PROGRAM OK_Repartiteurs_Laser
VAR
	B_820REP1: FB_Rep_Ethercat_MURR;
	B_821REP1: FB_Rep_Ethercat_MURR;
	B_822REP1: FB_Rep_Ethercat_MURR;
	Bandeaux_Leds: FB_LED_LC25C;
	Mesure_Presseur_Aval_Ref: FB_IOLink_Leuze_ODT3CL1;
	Mesure_Presseur_Aval_Opp_Ref: FB_IOLink_Leuze_ODT3CL1;
	Mesure_Presseur_Amont_Ref: FB_IOLink_Leuze_ODT3CL1;
	Mesure_Presseur_Amont_Opp_Ref: FB_IOLink_Leuze_ODT3CL1;
	FB_Servovanne_Gaz_TeteLaser: FB_IOLink_Servo_ITV2030;
	
	Txt_Alarme_Vanne,
	Txt_Defaut_Vanne	:STRING;
	
	Verrine_Machine			:FB_LED_LC25C;

	ReserveIOLink	:BOOL;
	
END_VAR

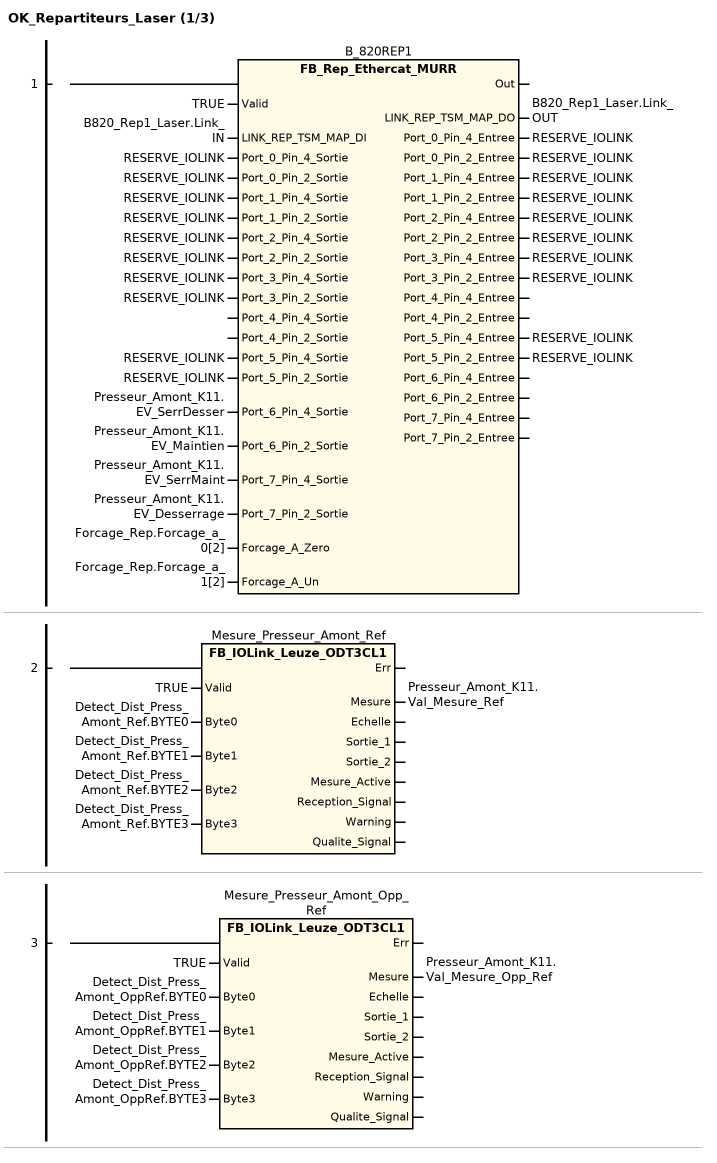
// NETWORK 1
B_820REP1(
    Valid := TRUE,
    LINK_REP_TSM_MAP_DI := B820_Rep1_Laser.Link_IN,
    Port_0_Pin_4_Sortie := RESERVE_IOLINK,
    Port_0_Pin_2_Sortie := RESERVE_IOLINK,
    Port_1_Pin_4_Sortie := RESERVE_IOLINK,
    Port_1_Pin_2_Sortie := RESERVE_IOLINK,
    Port_2_Pin_4_Sortie := RESERVE_IOLINK,
    Port_2_Pin_2_Sortie := RESERVE_IOLINK,
    Port_3_Pin_4_Sortie := RESERVE_IOLINK,
    Port_3_Pin_2_Sortie := RESERVE_IOLINK,
    Port_5_Pin_4_Sortie := RESERVE_IOLINK,
    Port_5_Pin_2_Sortie := RESERVE_IOLINK,
    Port_6_Pin_4_Sortie := Presseur_Amont_K11.EV_SerrDesser,
    Port_6_Pin_2_Sortie := Presseur_Amont_K11.EV_Maintien,
    Port_7_Pin_4_Sortie := Presseur_Amont_K11.EV_SerrMaint,
    Port_7_Pin_2_Sortie := Presseur_Amont_K11.EV_Desserrage,
    Forcage_A_Zero := Forcage_Rep.Forcage_a_0[2],
    Forcage_A_Un := Forcage_Rep.Forcage_a_1[2],
    LINK_REP_TSM_MAP_DO => B820_Rep1_Laser.Link_OUT,
    Port_0_Pin_4_Entree => RESERVE_IOLINK,
    Port_0_Pin_2_Entree => RESERVE_IOLINK,
    Port_1_Pin_4_Entree => RESERVE_IOLINK,
    Port_1_Pin_2_Entree => RESERVE_IOLINK,
    Port_2_Pin_4_Entree => RESERVE_IOLINK,
    Port_2_Pin_2_Entree => RESERVE_IOLINK,
    Port_3_Pin_4_Entree => RESERVE_IOLINK,
    Port_3_Pin_2_Entree => RESERVE_IOLINK,
    Port_5_Pin_4_Entree => RESERVE_IOLINK,
    Port_5_Pin_2_Entree => RESERVE_IOLINK); // FB_Rep_Ethercat_MURR

// NETWORK 2
Mesure_Presseur_Amont_Ref(
    Valid := TRUE,
    Byte0 := Detect_Dist_Press_Amont_Ref.BYTE0,
    Byte1 := Detect_Dist_Press_Amont_Ref.BYTE1,
    Byte2 := Detect_Dist_Press_Amont_Ref.BYTE2,
    Byte3 := Detect_Dist_Press_Amont_Ref.BYTE3,
    Mesure => Presseur_Amont_K11.Val_Mesure_Ref); // FB_IOLink_Leuze_ODT3CL1

// NETWORK 3
Mesure_Presseur_Amont_Opp_Ref(
    Valid := TRUE,
    Byte0 := Detect_Dist_Press_Amont_OppRef.BYTE0,
    Byte1 := Detect_Dist_Press_Amont_OppRef.BYTE1,
    Byte2 := Detect_Dist_Press_Amont_OppRef.BYTE2,
    Byte3 := Detect_Dist_Press_Amont_OppRef.BYTE3,
    Mesure => Presseur_Amont_K11.Val_Mesure_Opp_Ref); // FB_IOLink_Leuze_ODT3CL1

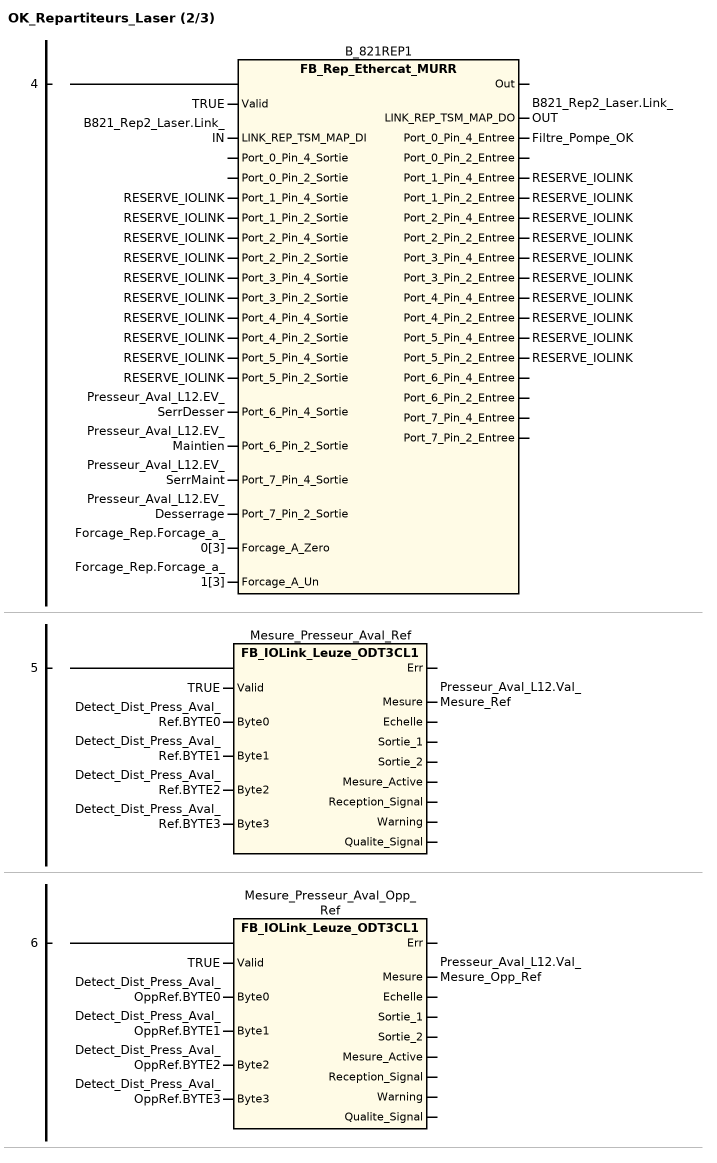
// NETWORK 4
B_821REP1(
    Valid := TRUE,
    LINK_REP_TSM_MAP_DI := B821_Rep2_Laser.Link_IN,
    Port_1_Pin_4_Sortie := RESERVE_IOLINK,
    Port_1_Pin_2_Sortie := RESERVE_IOLINK,
    Port_2_Pin_4_Sortie := RESERVE_IOLINK,
    Port_2_Pin_2_Sortie := RESERVE_IOLINK,
    Port_3_Pin_4_Sortie := RESERVE_IOLINK,
    Port_3_Pin_2_Sortie := RESERVE_IOLINK,
    Port_4_Pin_4_Sortie := RESERVE_IOLINK,
    Port_4_Pin_2_Sortie := RESERVE_IOLINK,
    Port_5_Pin_4_Sortie := RESERVE_IOLINK,
    Port_5_Pin_2_Sortie := RESERVE_IOLINK,
    Port_6_Pin_4_Sortie := Presseur_Aval_L12.EV_SerrDesser,
    Port_6_Pin_2_Sortie := Presseur_Aval_L12.EV_Maintien,
    Port_7_Pin_4_Sortie := Presseur_Aval_L12.EV_SerrMaint,
    Port_7_Pin_2_Sortie := Presseur_Aval_L12.EV_Desserrage,
    Forcage_A_Zero := Forcage_Rep.Forcage_a_0[3],
    Forcage_A_Un := Forcage_Rep.Forcage_a_1[3],
    LINK_REP_TSM_MAP_DO => B821_Rep2_Laser.Link_OUT,
    Port_0_Pin_4_Entree => Filtre_Pompe_OK,
    Port_1_Pin_4_Entree => RESERVE_IOLINK,
    Port_1_Pin_2_Entree => RESERVE_IOLINK,
    Port_2_Pin_4_Entree => RESERVE_IOLINK,
    Port_2_Pin_2_Entree => RESERVE_IOLINK,
    Port_3_Pin_4_Entree => RESERVE_IOLINK,
    Port_3_Pin_2_Entree => RESERVE_IOLINK,
    Port_4_Pin_4_Entree => RESERVE_IOLINK,
    Port_4_Pin_2_Entree => RESERVE_IOLINK,
    Port_5_Pin_4_Entree => RESERVE_IOLINK,
    Port_5_Pin_2_Entree => RESERVE_IOLINK); // FB_Rep_Ethercat_MURR

// NETWORK 5
Mesure_Presseur_Aval_Ref(
    Valid := TRUE,
    Byte0 := Detect_Dist_Press_Aval_Ref.BYTE0,
    Byte1 := Detect_Dist_Press_Aval_Ref.BYTE1,
    Byte2 := Detect_Dist_Press_Aval_Ref.BYTE2,
    Byte3 := Detect_Dist_Press_Aval_Ref.BYTE3,
    Mesure => Presseur_Aval_L12.Val_Mesure_Ref); // FB_IOLink_Leuze_ODT3CL1

// NETWORK 6
Mesure_Presseur_Aval_Opp_Ref(
    Valid := TRUE,
    Byte0 := Detect_Dist_Press_Aval_OppRef.BYTE0,
    Byte1 := Detect_Dist_Press_Aval_OppRef.BYTE1,
    Byte2 := Detect_Dist_Press_Aval_OppRef.BYTE2,
    Byte3 := Detect_Dist_Press_Aval_OppRef.BYTE3,
    Mesure => Presseur_Aval_L12.Val_Mesure_Opp_Ref); // FB_IOLink_Leuze_ODT3CL1

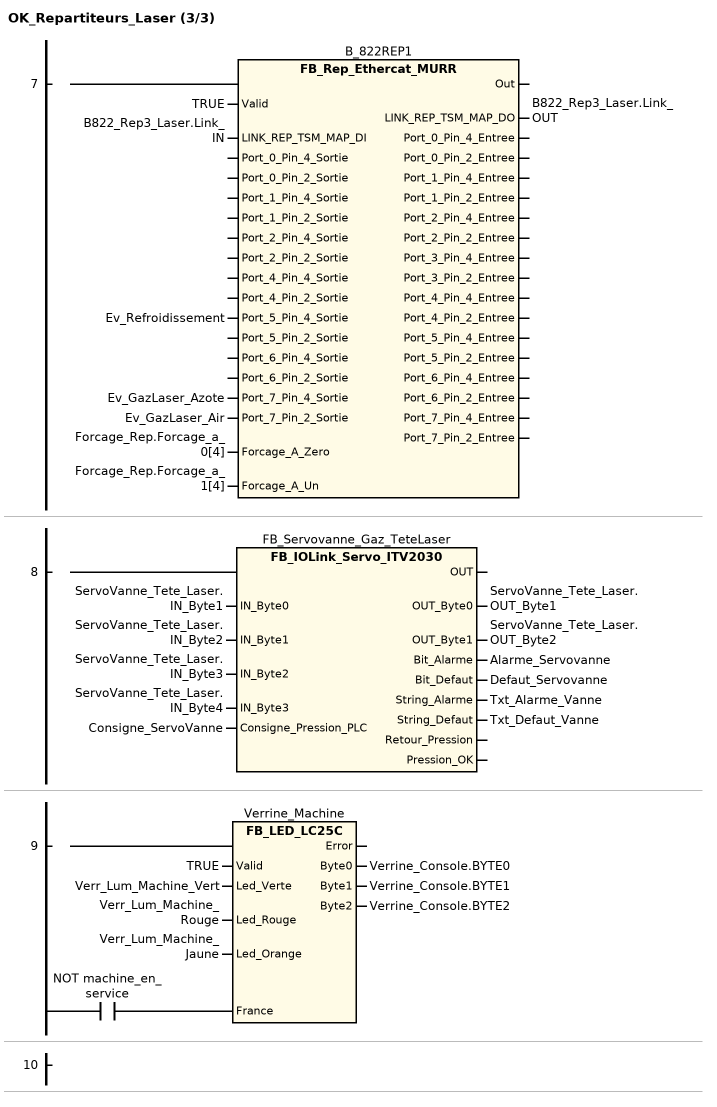
// NETWORK 7
B_822REP1(
    Valid := TRUE,
    LINK_REP_TSM_MAP_DI := B822_Rep3_Laser.Link_IN,
    Port_5_Pin_4_Sortie := Ev_Refroidissement,
    Port_7_Pin_4_Sortie := Ev_GazLaser_Azote,
    Port_7_Pin_2_Sortie := Ev_GazLaser_Air,
    Forcage_A_Zero := Forcage_Rep.Forcage_a_0[4],
    Forcage_A_Un := Forcage_Rep.Forcage_a_1[4],
    LINK_REP_TSM_MAP_DO => B822_Rep3_Laser.Link_OUT); // FB_Rep_Ethercat_MURR

// NETWORK 8
FB_Servovanne_Gaz_TeteLaser(
    IN_Byte0 := ServoVanne_Tete_Laser.IN_Byte1,
    IN_Byte1 := ServoVanne_Tete_Laser.IN_Byte2,
    IN_Byte2 := ServoVanne_Tete_Laser.IN_Byte3,
    IN_Byte3 := ServoVanne_Tete_Laser.IN_Byte4,
    Consigne_Pression_PLC := Consigne_ServoVanne,
    OUT_Byte0 => ServoVanne_Tete_Laser.OUT_Byte1,
    OUT_Byte1 => ServoVanne_Tete_Laser.OUT_Byte2,
    Bit_Alarme => Alarme_Servovanne,
    Bit_Defaut => Defaut_Servovanne,
    String_Alarme => Txt_Alarme_Vanne,
    String_Defaut => Txt_Defaut_Vanne); // FB_IOLink_Servo_ITV2030

// NETWORK 9
Verrine_Machine(
    Valid := TRUE,
    Led_Verte := Verr_Lum_Machine_Vert,
    Led_Rouge := Verr_Lum_Machine_Rouge,
    Led_Orange := Verr_Lum_Machine_Jaune,
    France := NOT machine_en_service,
    Byte0 => Verrine_Console.BYTE0,
    Byte1 => Verrine_Console.BYTE1,
    Byte2 => Verrine_Console.BYTE2); // FB_LED_LC25C

// NETWORK 10

END_PROGRAM

(* stored: Version 1.1.0.1
   POU OK_Repartiteurs_Laser: Id {be51289f-c5e6-4098-9d9a-63a509403054}, SpecialFunc None *)
